
TYPE "Config_001"
STRUCT
        DINT_VAL : INT;
        INT_ARRAY : ARRAY[0..10] OF INT;
        REAL_ARRAY : ARRAY[0..10] OF REAL;
END_STRUCT;
END_TYPE